{attribute 'linkalways'} 
{attribute 'no_explicit_call' := 'This FB is a CLASS and must be accessed using methods or properties'}
{attribute 'enable_dynamic_creation'}
FUNCTION_BLOCK FINAL MAX_LWORD EXTENDS Node
VAR
	in1 : _LWORD(0);
	in2 : _LWORD(0);
	out : _LWORD(0);
END_VAR

METHOD PUBLIC Clone : I_Node
VAR
	pNode : POINTER TO MAX_LWORD;
END_VAR
pNode := __NEW(MAX_LWORD);
Clone := pNode^;
END_METHOD

METHOD FB_init : BOOL
VAR_INPUT
	bInitRetains : BOOL; // if TRUE, the retain variables are initialized (warm start / cold start)
	bInCopyCode : BOOL;  // if TRUE, the instance afterwards gets moved into the copy code (online change)
END_VAR
AddInput('in1',THIS^.in1);
AddInput('in2',THIS^.in2);
AddOutput('out', THIS^.out);
END_METHOD

METHOD PROTECTED OnExecute
VAR
END_VAR
out.Value := MAX(in1.Value, in2.Value);
END_METHOD

END_FUNCTION_BLOCK

(* stored: Version 1.1.0.1, ProductVersion 3.1.4024.15
   POU MAX_LWORD: Id {ac646771-299e-4d3c-960c-4de5c2e1609b}, SpecialFunc None
   Folder Constructor: Id {d8016430-b454-4911-8fd6-d30b590ba9ab}
   Method Clone: Id {6c7af5d3-036f-458c-9df3-cad143c6dc5a}
   Method FB_init: Id {c3cc5ea9-9ee9-44ad-9ad5-40a74e263cfd}
   Method OnExecute: Id {b41a22b6-4699-4d90-8a03-3001dc70db9f} *)
